// Mitsubishi GX Works2 project: Jesús Beato 2023-1283 #4   PLC: FX2N/FX2NC

PROGRAM MAIN
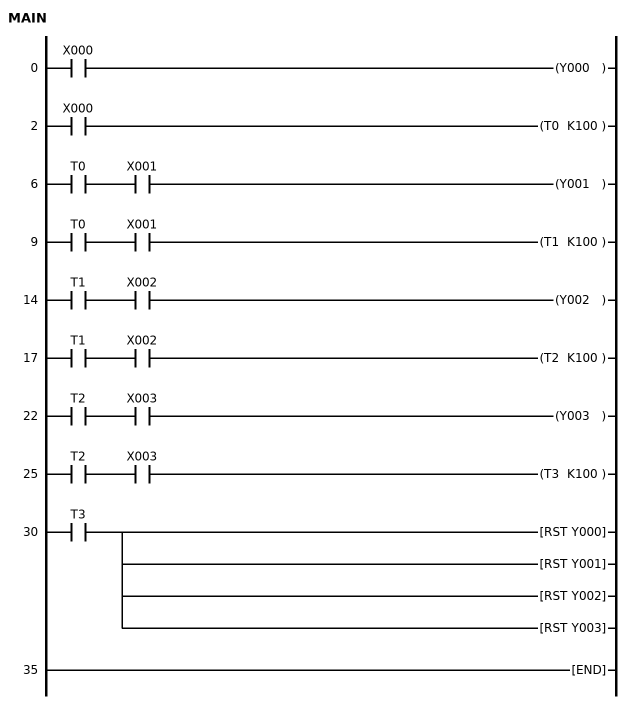
0     LD      X000
      OUT     Y000
2     LD      X000
      OUT     T0 K100
6     LD      T0
      AND     X001
      OUT     Y001
9     LD      T0
      AND     X001
      OUT     T1 K100
14    LD      T1
      AND     X002
      OUT     Y002
17    LD      T1
      AND     X002
      OUT     T2 K100
22    LD      T2
      AND     X003
      OUT     Y003
25    LD      T2
      AND     X003
      OUT     T3 K100
30    LD      T3
      RST     Y000
      RST     Y001
      RST     Y002
      RST     Y003
35    END
END_PROGRAM
